% RSLogix 500 project BAW TYK 3 (2).RSS, saved by version 8.40.00.08 %
PROJECT "UNTITLED"    % processor: type code 33 %

PROGRAM FILES
  LAD 2   3 rungs

DATA FILES
  S2 STATUS  164 elements
  B3 BINARY  1 elements
  T4 TIMER  1 elements
  C5 COUNTER  1 elements
  R6 CONTROL  1 elements
  N7 INTEGER  1 elements
  F8 FLOAT  1 elements

LADDER 2
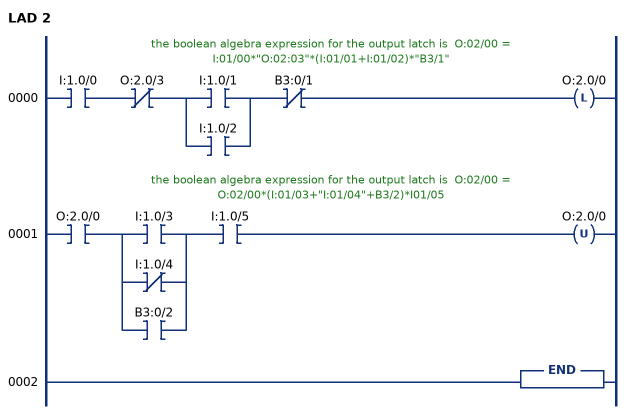
% Rung: 0 %  % edit flag set %
% the boolean algebra expression for the output latch is  O:02/00 = I:01/00*"O:02:03"*(I:01/01+I:01/02)*"B3/1" %
SOR XIC I:1.0/0 XIO O:2.0/3 BST XIC I:1.0/1 NXB XIC I:1.0/2 BND XIO B3:0/1 OTL O:2.0/0 EOR
% Rung: 1 %  % edit flag set %
% the boolean algebra expression for the output latch is  O:02/00 = O:02/00*(I:01/03+"I:01/04"+B3/2)*I01/05 %
SOR XIC O:2.0/0 BST XIC I:1.0/3 NXB BST XIO I:1.0/4 NXB XIC B3:0/2 BND BND XIC I:1.0/5 OTU O:2.0/0 EOR
% Rung: 2 %
SOR END EOR
